INTERFACE ITFGesimuleerdDI

PROPERTY SensorWaarde : bool
GET
END_GET
SET
END_SET
END_PROPERTY

END_INTERFACE

(* stored: Version 1.1.0.1
   Itf ITFGesimuleerdDI: Id {78acb92f-277c-4702-b5bd-e92f97d32b4b}
   Property SensorWaarde: Id {beead022-26ca-4709-af0f-7fabe318762d}
   Get Get: Id {0326520b-45ca-4bae-9787-a725827f190b}
   Set Set: Id {0aba72d5-1aaf-4a07-a927-834466809ca2} *)
